# EPICS autosave request: iocs/pvcamIOC/iocBoot/ioc16PvCam/auto_settings.req
file "pvCam_settings.req",  	    P=$(P),  R=cam1:
file "NDStdArrays_settings.req",  P=$(P),  R=image1:
file "commonPlugin_settings.req", P=$(P)
